// TIA Portal V18 export
DATA_BLOCK "ST10_FB_S7connect_IDB"   // DB900
// stored: AutoNumber false, InstanceOfName ST10_FB_S7connect, InstanceOfType FB
"ST10_FB_S7connect"
   // VAR_INPUT
   //    "CLOCK_0.2_SEC" : Bool;
   // END_VAR
   // VAR
   //    Always_On : Bool;
   //    Status_Get : Array[1..6] of Struct
   //       NDR : Bool;
   //       Error : Bool;
   //       Status : Int;
   //    END_STRUCT;
   //    Status_Put : Array[1..6] of Struct
   //       Done : Bool;
   //       Error : Bool;
   //       Status : Int;
   //    END_STRUCT;
   //    GET_Instance1 { S7_SetPoint := 'True'} : GET;
   //    GET_Instance2 { S7_SetPoint := 'True'} : GET;
   //    PUT_Instance1 { S7_SetPoint := 'True'} : PUT;
   //    PUT_Instance2 { S7_SetPoint := 'True'} : PUT;
   //    PLs { S7_SetPoint := 'True'} : Array[1..6] of Bool;
   //    TON : Array[1..5] of TON_TIME;
   //    NextStation_OffLine : Bool;
   // END_VAR
BEGIN
END_DATA_BLOCK
